//----------------------------------------------------------------------------//
//            Copyright 2018 Rieckermann Engineering Operations               //
//----------------------------------------------------------------------------//
// Class:       fcHMIInterfaceBLK                                             //
// Description:                                                               //
// Manages the data interface for the HMI BLK faceplate.                      //
//----------------------------------------------------------------------------//
// Revision history:                                                          //
// Rev By               Date        CC        Note                            //
// 2.0 David Paspa      03-Aug-2018 NA        Reboot for S7-1500.             //
// 0.1 Khairul Basar    03-Aug-2009           Initial design.                 //
//----------------------------------------------------------------------------//
FUNCTION "fcHMIInterfaceBLK" : Void
TITLE = HMI BLK Faceplate interface
{ S7_Optimized_Access := 'FALSE' }
AUTHOR : REO
NAME : fcHMIInterfaceBLK
VERSION : 2.0

//----------------------------------------------------------------------------//
// Declare interface and variables:                                           //
//----------------------------------------------------------------------------//
VAR_IN_OUT
    bmc : "udtModeCommandBLK"; // Block events
    err : "udtBLKError";       // Block error
    mcr : "udtMCRead";         // Block read mode and command
    mcw : "udtMCWrite";        // Block write mode and command
END_VAR

VAR_TEMP
    outAUTO : Bool;
    retVal : Int;
END_VAR

BEGIN
NETWORK
TITLE = Copy the BLK event data to the HMI interface block
    //------------------------------------------------------------------------//
    // Copy BLK event data:                                                   //
    //------------------------------------------------------------------------//
    CALL BLKMOV
    {blk_type := 'Any'}
    (   SRCBLK               := #bmc ,
        RET_VAL              := #retVal ,
        DSTBLK               := "dbHMIInterfaceBLK".buffer.block.bmc
    );

NETWORK
TITLE = Copy the BLK error data to the HMI interface block
    //------------------------------------------------------------------------//
    // Copy BLK event data:                                                   //
    //------------------------------------------------------------------------//
    CALL BLKMOV
    {blk_type := 'Any'}
    (   SRCBLK               := #err ,
        RET_VAL              := #retVal ,
        DSTBLK               := "dbHMIInterfaceBLK".buffer.block.err
    );

NETWORK
TITLE = Copy the BLK read mode and command data to the HMI interface block
    //------------------------------------------------------------------------//
    // Copy read mode and command data:                                     //
    //------------------------------------------------------------------------//
    CALL BLKMOV
    {blk_type := 'Any'}
    (   SRCBLK               := #mcr ,
        RET_VAL              := #retVal ,
        DSTBLK               := "dbHMIInterfaceBLK".buffer.block.mcr
    );

NETWORK
TITLE = Copy the BLK write mode and command data to the HMI interface block
    //------------------------------------------------------------------------//
    // Copy write mode and command data:                                      //
    //------------------------------------------------------------------------//
    CALL BLKMOV
    {blk_type := 'Any'}
    (   SRCBLK               := #mcw ,
        RET_VAL              := #retVal ,
        DSTBLK               := "dbHMIInterfaceBLK".buffer.block.mcw
    );

END_FUNCTION
